// TIA Portal V17 export
// export: Created 2022-07-16T16:56:14.5326582Z, ExportSetting WithDefaults, DisplayName Totally Integrated Automation Portal, DisplayVersion V17, DisplayName TIA Portal Openness, DisplayVersion V17, DisplayName TIA Portal Version Control Interface, DisplayVersion V17, DisplayName TIA Portal Test Suite Advanced, DisplayVersion V17, DisplayName STEP 7 Professional, DisplayVersion V17, DisplayName STEP 7 Safety, DisplayVersion V17, DisplayName WinCC Professional, DisplayVersion V17
TYPE "Client interface_1.udtOtherPressure"
// stored: IsFailsafeCompliant false
   STRUCT
      avaragePressure { ExternalWritable := 'False'} : Int;
      tripleValidationActive { ExternalWritable := 'False'} : Int;
      dualValidationActive { ExternalWritable := 'False'} : Int;
      pressure1failed { ExternalWritable := 'False'} : Bool;
      pressure2failed { ExternalWritable := 'False'} : Bool;
      pressure3failed { ExternalWritable := 'False'} : Bool;
      moreThen1pressureFailed { ExternalWritable := 'False'} : Bool;
   END_STRUCT;
END_TYPE
